// TIA Portal V15.1 export
// export: Created 2024-05-17T05:38:58.6337777Z, ExportSetting WithDefaults, DisplayName Totally Integrated Automation Portal, DisplayVersion V15.1 Update 5, DisplayName TIA Portal Openness, DisplayVersion V15.1 Update 5, DisplayName SINAMICS Startdrive Advanced, DisplayVersion V15.1, DisplayName G130, G150, S120, S150, SINAMICS MV, S210, DisplayVersion V15.1, DisplayName G110M, G120, G120C, G120D, G120P, DisplayVersion V15.1, DisplayName STEP 7 Professional, DisplayVersion V15.1 Update 5, DisplayName STEP 7 Safety, DisplayVersion V15.1, DisplayName WinCC Professional, DisplayVersion V15.1 Update 5, DisplayName SIMATIC Visualization Architect, DisplayVersion V15.1
FUNCTION "209230ZS01AEAK" : Void   // FC421, FBD
TITLE = 209230ZS01AEAK
{ S7_Optimized_Access := 'TRUE' }
AUTHOR : VCC
VERSION : 0.1
// stored: AutoNumber false, IsIECCheckEnabled false, SetENOAutomatically False, UDAEnableTagReadback false
   VAR_OUTPUT
      O_AlarmA : Bool;   // Alarm A
      O_AlarmB : Bool;   // Alarm B
      O_AlarmC : Bool;   // Alarm C
      O_AlarmD : Bool;   // Alarm D
      O_AlarmABCondition : Bool;   // Alarm AB condition
      H_IAnim : Word;   // For animation of icon
   END_VAR
BEGIN

REGION Network 1: **** --------------------- AE01 --------------------- ****
END_REGION

REGION Network 2: **** 2.2 Alarms - Alarm generation **** AE01E3FS13 // CH1 - 24VDC Fuse - ModeZone230 - Switch / Busnode 230AX01 & 230AS10
   // 24VDC Fuse - ModeZone230 - Switch / Busnode 230AX01 & 230AS10
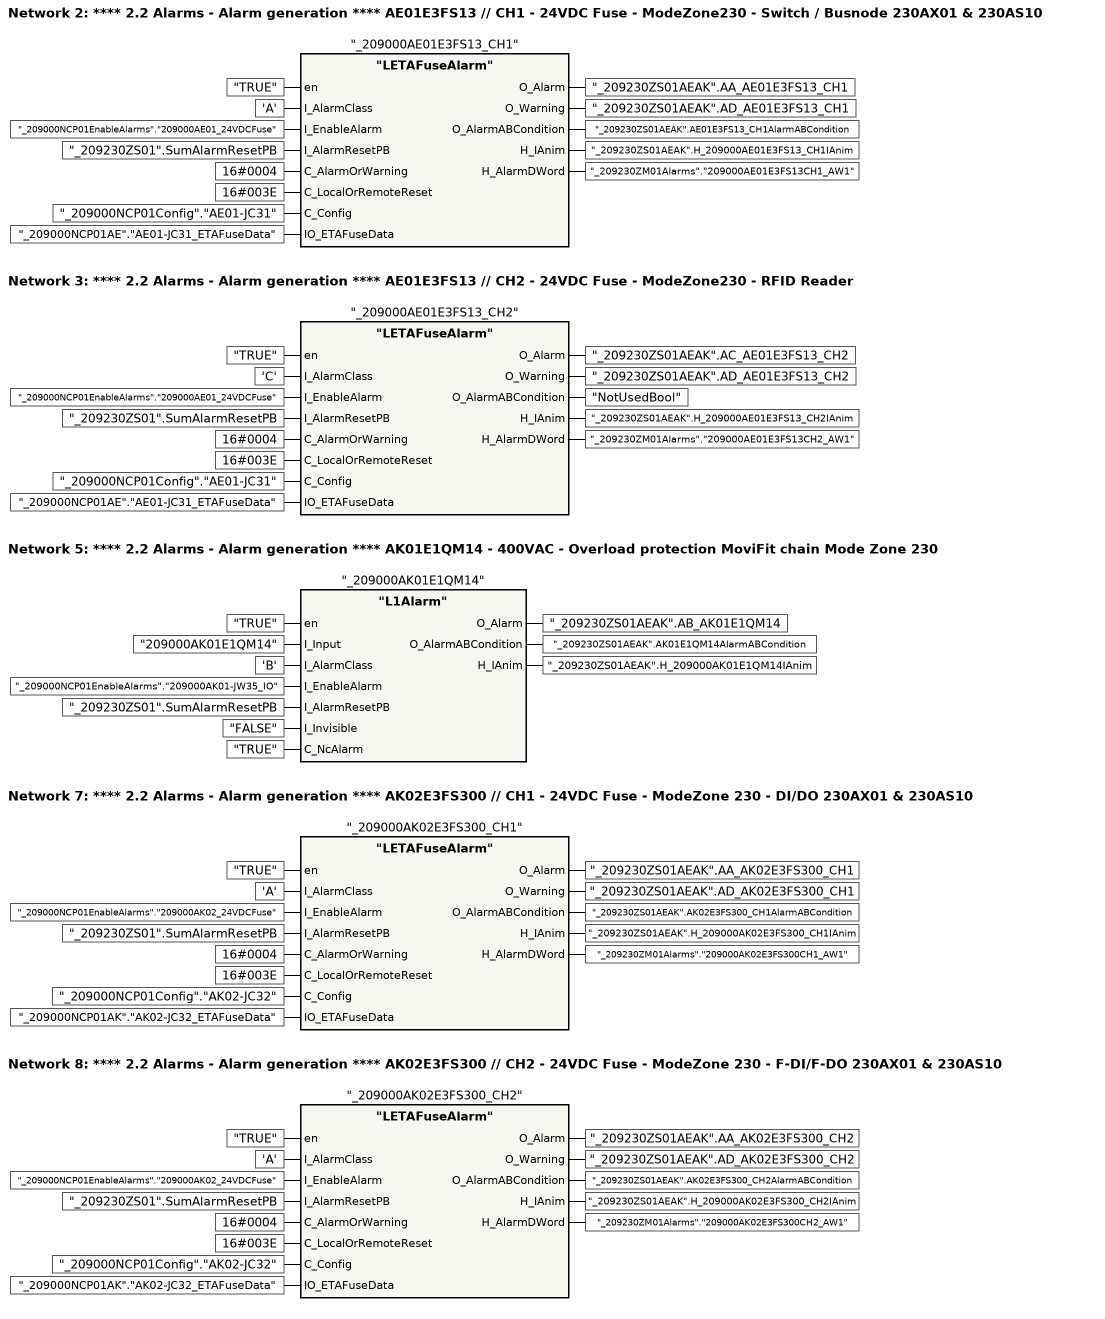
   IF "TRUE" THEN
       "_209000AE01E3FS13_CH1"(I_AlarmClass := 'A',   // "LETAFuseAlarm"
                               I_EnableAlarm := "_209000NCP01EnableAlarms"."209000AE01_24VDCFuse",
                               I_AlarmResetPB := "_209230ZS01".SumAlarmResetPB,
                               C_AlarmOrWarning := 16#0004,
                               C_LocalOrRemoteReset := 16#003E,
                               C_Config := "_209000NCP01Config"."AE01-JC31",
                               IO_ETAFuseData := "_209000NCP01AE"."AE01-JC31_ETAFuseData",
                               O_Alarm => "_209230ZS01AEAK".AA_AE01E3FS13_CH1,
                               O_Warning => "_209230ZS01AEAK".AD_AE01E3FS13_CH1,
                               O_AlarmABCondition => "_209230ZS01AEAK".AE01E3FS13_CH1AlarmABCondition,
                               H_IAnim => "_209230ZS01AEAK".H_209000AE01E3FS13_CH1IAnim,
                               H_AlarmDWord => "_209230ZM01Alarms"."209000AE01E3FS13CH1_AW1");
   END_IF;
END_REGION

REGION Network 3: **** 2.2 Alarms - Alarm generation **** AE01E3FS13 // CH2 - 24VDC Fuse - ModeZone230 - RFID Reader
   // 24VDC Fuse - ModeZone230 - RFID Reader
   IF "TRUE" THEN
       "_209000AE01E3FS13_CH2"(I_AlarmClass := 'C',   // "LETAFuseAlarm"
                               I_EnableAlarm := "_209000NCP01EnableAlarms"."209000AE01_24VDCFuse",
                               I_AlarmResetPB := "_209230ZS01".SumAlarmResetPB,
                               C_AlarmOrWarning := 16#0004,
                               C_LocalOrRemoteReset := 16#003E,
                               C_Config := "_209000NCP01Config"."AE01-JC31",
                               IO_ETAFuseData := "_209000NCP01AE"."AE01-JC31_ETAFuseData",
                               O_Alarm => "_209230ZS01AEAK".AC_AE01E3FS13_CH2,
                               O_Warning => "_209230ZS01AEAK".AD_AE01E3FS13_CH2,
                               O_AlarmABCondition => "NotUsedBool",
                               H_IAnim => "_209230ZS01AEAK".H_209000AE01E3FS13_CH2IAnim,
                               H_AlarmDWord => "_209230ZM01Alarms"."209000AE01E3FS13CH2_AW1");
   END_IF;
END_REGION

REGION Network 4: **** --------------------- AK01 --------------------- ****
END_REGION

REGION Network 5: **** 2.2 Alarms - Alarm generation **** AK01E1QM14 - 400VAC - Overload protection MoviFit chain Mode Zone 230
   // 400VAC - Overload protection MoviFit chain Mode Zone 230
   IF "TRUE" THEN
       "_209000AK01E1QM14"(I_Input := "209000AK01E1QM14",   // "L1Alarm"
                           I_AlarmClass := 'B',
                           I_EnableAlarm := "_209000NCP01EnableAlarms"."209000AK01-JW35_IO",
                           I_AlarmResetPB := "_209230ZS01".SumAlarmResetPB,
                           I_Invisible := "FALSE",
                           C_NcAlarm := "TRUE",
                           O_Alarm => "_209230ZS01AEAK".AB_AK01E1QM14,
                           O_AlarmABCondition => "_209230ZS01AEAK".AK01E1QM14AlarmABCondition,
                           H_IAnim => "_209230ZS01AEAK".H_209000AK01E1QM14IAnim);
   END_IF;
END_REGION

REGION Network 6: **** --------------------- AK02 --------------------- ****
END_REGION

REGION Network 7: **** 2.2 Alarms - Alarm generation **** AK02E3FS300 // CH1 - 24VDC Fuse - ModeZone 230 - DI/DO 230AX01 & 230AS10
   // 24VDC Fuse - ModeZone 230 - DI/DO 230AX01 & 230AS10
   IF "TRUE" THEN
       "_209000AK02E3FS300_CH1"(I_AlarmClass := 'A',   // "LETAFuseAlarm"
                               I_EnableAlarm := "_209000NCP01EnableAlarms"."209000AK02_24VDCFuse",
                               I_AlarmResetPB := "_209230ZS01".SumAlarmResetPB,
                               C_AlarmOrWarning := 16#0004,
                               C_LocalOrRemoteReset := 16#003E,
                               C_Config := "_209000NCP01Config"."AK02-JC32",
                               IO_ETAFuseData := "_209000NCP01AK"."AK02-JC32_ETAFuseData",
                               O_Alarm => "_209230ZS01AEAK".AA_AK02E3FS300_CH1,
                               O_Warning => "_209230ZS01AEAK".AD_AK02E3FS300_CH1,
                               O_AlarmABCondition => "_209230ZS01AEAK".AK02E3FS300_CH1AlarmABCondition,
                               H_IAnim => "_209230ZS01AEAK".H_209000AK02E3FS300_CH1IAnim,
                               H_AlarmDWord => "_209230ZM01Alarms"."209000AK02E3FS300CH1_AW1");
   END_IF;
END_REGION

REGION Network 8: **** 2.2 Alarms - Alarm generation **** AK02E3FS300 // CH2 - 24VDC Fuse - ModeZone 230 - F-DI/F-DO 230AX01 & 230AS10
   // 24VDC Fuse - ModeZone 230 - F-DI/F-DO 230AX01 & 230AS10
   IF "TRUE" THEN
       "_209000AK02E3FS300_CH2"(I_AlarmClass := 'A',   // "LETAFuseAlarm"
                               I_EnableAlarm := "_209000NCP01EnableAlarms"."209000AK02_24VDCFuse",
                               I_AlarmResetPB := "_209230ZS01".SumAlarmResetPB,
                               C_AlarmOrWarning := 16#0004,
                               C_LocalOrRemoteReset := 16#003E,
                               C_Config := "_209000NCP01Config"."AK02-JC32",
                               IO_ETAFuseData := "_209000NCP01AK"."AK02-JC32_ETAFuseData",
                               O_Alarm => "_209230ZS01AEAK".AA_AK02E3FS300_CH2,
                               O_Warning => "_209230ZS01AEAK".AD_AK02E3FS300_CH2,
                               O_AlarmABCondition => "_209230ZS01AEAK".AK02E3FS300_CH2AlarmABCondition,
                               H_IAnim => "_209230ZS01AEAK".H_209000AK02E3FS300_CH2IAnim,
                               H_AlarmDWord => "_209230ZM01Alarms"."209000AK02E3FS300CH2_AW1");
   END_IF;
END_REGION

REGION Network 9: **** 2.2 Alarms - Alarm generation **** AK02E3FS301 // CH1 - 24VDC Fuse - ModeZone 230 - Doorlock
   // 24VDC Fuse - ModeZone 230 - Doorlock
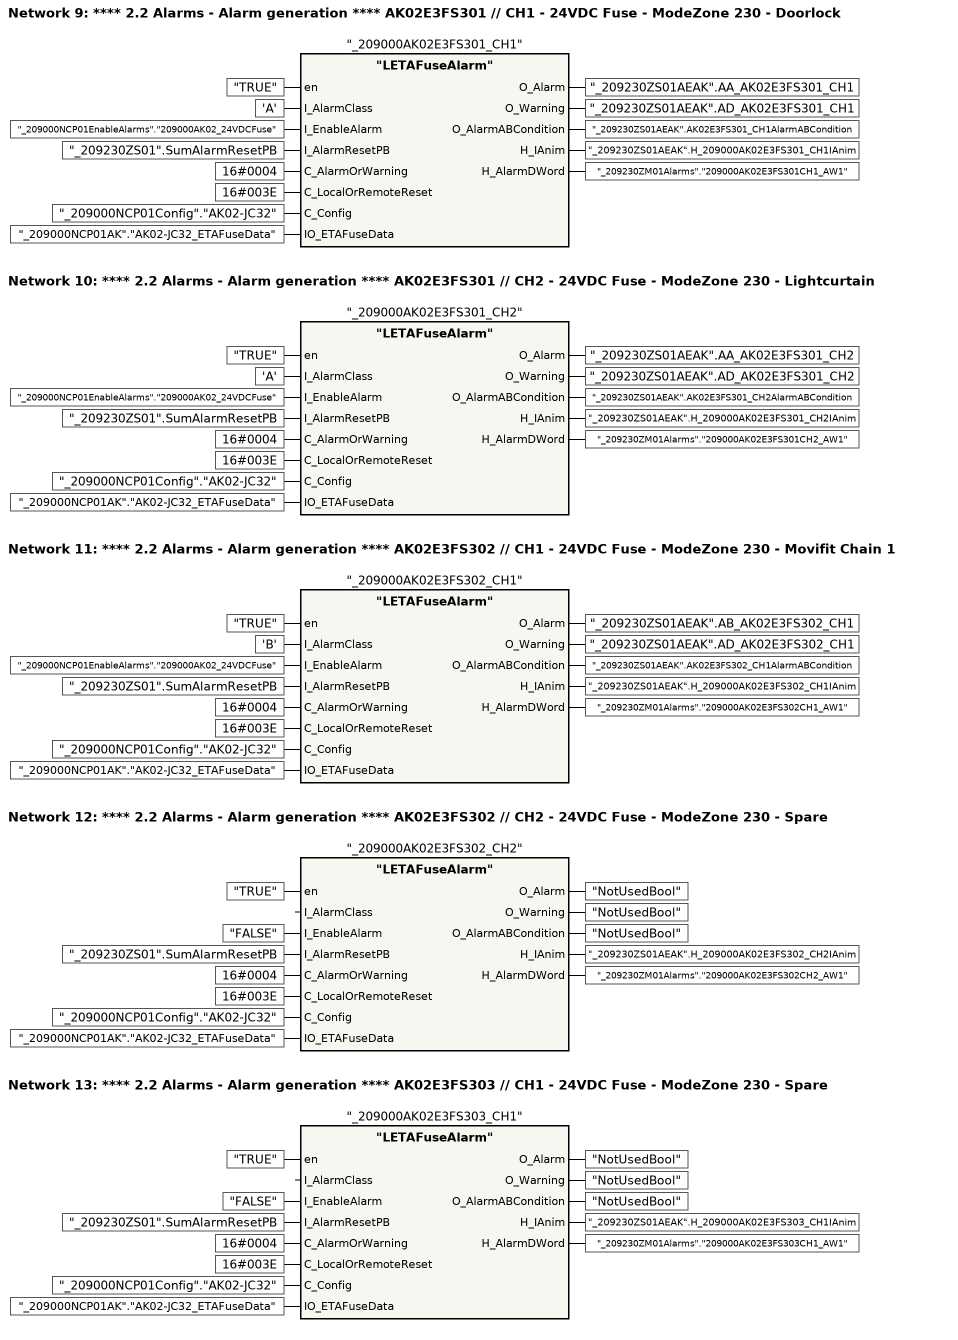
   IF "TRUE" THEN
       "_209000AK02E3FS301_CH1"(I_AlarmClass := 'A',   // "LETAFuseAlarm"
                               I_EnableAlarm := "_209000NCP01EnableAlarms"."209000AK02_24VDCFuse",
                               I_AlarmResetPB := "_209230ZS01".SumAlarmResetPB,
                               C_AlarmOrWarning := 16#0004,
                               C_LocalOrRemoteReset := 16#003E,
                               C_Config := "_209000NCP01Config"."AK02-JC32",
                               IO_ETAFuseData := "_209000NCP01AK"."AK02-JC32_ETAFuseData",
                               O_Alarm => "_209230ZS01AEAK".AA_AK02E3FS301_CH1,
                               O_Warning => "_209230ZS01AEAK".AD_AK02E3FS301_CH1,
                               O_AlarmABCondition => "_209230ZS01AEAK".AK02E3FS301_CH1AlarmABCondition,
                               H_IAnim => "_209230ZS01AEAK".H_209000AK02E3FS301_CH1IAnim,
                               H_AlarmDWord => "_209230ZM01Alarms"."209000AK02E3FS301CH1_AW1");
   END_IF;
END_REGION

REGION Network 10: **** 2.2 Alarms - Alarm generation **** AK02E3FS301 // CH2 - 24VDC Fuse - ModeZone 230 - Lightcurtain
   // 24VDC Fuse - ModeZone 230 - Lightcurtain
   IF "TRUE" THEN
       "_209000AK02E3FS301_CH2"(I_AlarmClass := 'A',   // "LETAFuseAlarm"
                               I_EnableAlarm := "_209000NCP01EnableAlarms"."209000AK02_24VDCFuse",
                               I_AlarmResetPB := "_209230ZS01".SumAlarmResetPB,
                               C_AlarmOrWarning := 16#0004,
                               C_LocalOrRemoteReset := 16#003E,
                               C_Config := "_209000NCP01Config"."AK02-JC32",
                               IO_ETAFuseData := "_209000NCP01AK"."AK02-JC32_ETAFuseData",
                               O_Alarm => "_209230ZS01AEAK".AA_AK02E3FS301_CH2,
                               O_Warning => "_209230ZS01AEAK".AD_AK02E3FS301_CH2,
                               O_AlarmABCondition => "_209230ZS01AEAK".AK02E3FS301_CH2AlarmABCondition,
                               H_IAnim => "_209230ZS01AEAK".H_209000AK02E3FS301_CH2IAnim,
                               H_AlarmDWord => "_209230ZM01Alarms"."209000AK02E3FS301CH2_AW1");
   END_IF;
END_REGION

REGION Network 11: **** 2.2 Alarms - Alarm generation **** AK02E3FS302 // CH1 - 24VDC Fuse - ModeZone 230 - Movifit Chain 1
   // 24VDC Fuse - ModeZone 230 - Movifit Chain 1
   IF "TRUE" THEN
       "_209000AK02E3FS302_CH1"(I_AlarmClass := 'B',   // "LETAFuseAlarm"
                               I_EnableAlarm := "_209000NCP01EnableAlarms"."209000AK02_24VDCFuse",
                               I_AlarmResetPB := "_209230ZS01".SumAlarmResetPB,
                               C_AlarmOrWarning := 16#0004,
                               C_LocalOrRemoteReset := 16#003E,
                               C_Config := "_209000NCP01Config"."AK02-JC32",
                               IO_ETAFuseData := "_209000NCP01AK"."AK02-JC32_ETAFuseData",
                               O_Alarm => "_209230ZS01AEAK".AB_AK02E3FS302_CH1,
                               O_Warning => "_209230ZS01AEAK".AD_AK02E3FS302_CH1,
                               O_AlarmABCondition => "_209230ZS01AEAK".AK02E3FS302_CH1AlarmABCondition,
                               H_IAnim => "_209230ZS01AEAK".H_209000AK02E3FS302_CH1IAnim,
                               H_AlarmDWord => "_209230ZM01Alarms"."209000AK02E3FS302CH1_AW1");
   END_IF;
END_REGION

REGION Network 12: **** 2.2 Alarms - Alarm generation **** AK02E3FS302 // CH2 - 24VDC Fuse - ModeZone 230 - Spare
   // 24VDC Fuse - ModeZone 230 - Spare
   IF "TRUE" THEN
       "_209000AK02E3FS302_CH2"(I_EnableAlarm := "FALSE",   // "LETAFuseAlarm"
                               I_AlarmResetPB := "_209230ZS01".SumAlarmResetPB,
                               C_AlarmOrWarning := 16#0004,
                               C_LocalOrRemoteReset := 16#003E,
                               C_Config := "_209000NCP01Config"."AK02-JC32",
                               IO_ETAFuseData := "_209000NCP01AK"."AK02-JC32_ETAFuseData",
                               O_Alarm => "NotUsedBool",
                               O_Warning => "NotUsedBool",
                               O_AlarmABCondition => "NotUsedBool",
                               H_IAnim => "_209230ZS01AEAK".H_209000AK02E3FS302_CH2IAnim,
                               H_AlarmDWord => "_209230ZM01Alarms"."209000AK02E3FS302CH2_AW1");
   END_IF;
END_REGION

REGION Network 13: **** 2.2 Alarms - Alarm generation **** AK02E3FS303 // CH1 - 24VDC Fuse - ModeZone 230 - Spare
   // 24VDC Fuse - ModeZone 230 - Spare
   IF "TRUE" THEN
       "_209000AK02E3FS303_CH1"(I_EnableAlarm := "FALSE",   // "LETAFuseAlarm"
                               I_AlarmResetPB := "_209230ZS01".SumAlarmResetPB,
                               C_AlarmOrWarning := 16#0004,
                               C_LocalOrRemoteReset := 16#003E,
                               C_Config := "_209000NCP01Config"."AK02-JC32",
                               IO_ETAFuseData := "_209000NCP01AK"."AK02-JC32_ETAFuseData",
                               O_Alarm => "NotUsedBool",
                               O_Warning => "NotUsedBool",
                               O_AlarmABCondition => "NotUsedBool",
                               H_IAnim => "_209230ZS01AEAK".H_209000AK02E3FS303_CH1IAnim,
                               H_AlarmDWord => "_209230ZM01Alarms"."209000AK02E3FS303CH1_AW1");
   END_IF;
END_REGION

REGION Network 14: **** 2.2 Alarms - Alarm generation **** AK02E3FS303 // CH2 - 24VDC Fuse - ModeZone 230 - Spare
   // 24VDC Fuse - ModeZone 230 - Spare
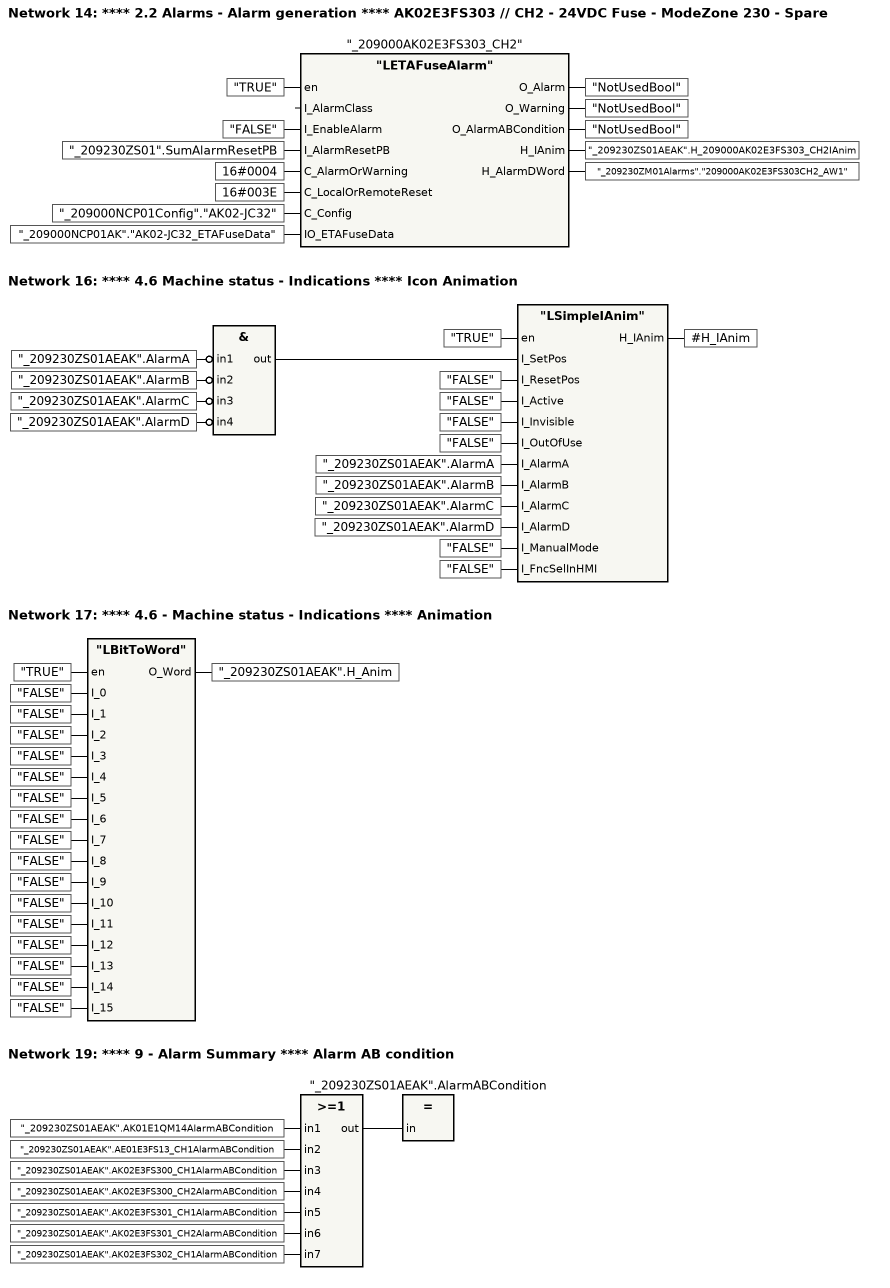
   IF "TRUE" THEN
       "_209000AK02E3FS303_CH2"(I_EnableAlarm := "FALSE",   // "LETAFuseAlarm"
                               I_AlarmResetPB := "_209230ZS01".SumAlarmResetPB,
                               C_AlarmOrWarning := 16#0004,
                               C_LocalOrRemoteReset := 16#003E,
                               C_Config := "_209000NCP01Config"."AK02-JC32",
                               IO_ETAFuseData := "_209000NCP01AK"."AK02-JC32_ETAFuseData",
                               O_Alarm => "NotUsedBool",
                               O_Warning => "NotUsedBool",
                               O_AlarmABCondition => "NotUsedBool",
                               H_IAnim => "_209230ZS01AEAK".H_209000AK02E3FS303_CH2IAnim,
                               H_AlarmDWord => "_209230ZM01Alarms"."209000AK02E3FS303CH2_AW1");
   END_IF;
END_REGION

REGION Network 15: **** -------------------------------------------------- ****
END_REGION

REGION Network 16: **** 4.6 Machine status - Indications **** Icon Animation
   // Animation for icon
   IF "TRUE" THEN
       "LSimpleIAnim"(I_SetPos := NOT "_209230ZS01AEAK".AlarmA AND NOT "_209230ZS01AEAK".AlarmB AND NOT "_209230ZS01AEAK".AlarmC AND NOT "_209230ZS01AEAK".AlarmD,
                      I_ResetPos := "FALSE",
                      I_Active := "FALSE",
                      I_Invisible := "FALSE",
                      I_OutOfUse := "FALSE",
                      I_AlarmA := "_209230ZS01AEAK".AlarmA,
                      I_AlarmB := "_209230ZS01AEAK".AlarmB,
                      I_AlarmC := "_209230ZS01AEAK".AlarmC,
                      I_AlarmD := "_209230ZS01AEAK".AlarmD,
                      I_ManualMode := "FALSE",
                      I_FncSelInHMI := "FALSE",
                      H_IAnim => #H_IAnim);
   END_IF;
END_REGION

REGION Network 17: **** 4.6 - Machine status - Indications **** Animation
   // Animation
   IF "TRUE" THEN
       "LBitToWord"(I_0 := "FALSE",
                    I_1 := "FALSE",
                    I_2 := "FALSE",
                    I_3 := "FALSE",
                    I_4 := "FALSE",
                    I_5 := "FALSE",
                    I_6 := "FALSE",
                    I_7 := "FALSE",
                    I_8 := "FALSE",
                    I_9 := "FALSE",
                    I_10 := "FALSE",
                    I_11 := "FALSE",
                    I_12 := "FALSE",
                    I_13 := "FALSE",
                    I_14 := "FALSE",
                    I_15 := "FALSE",
                    O_Word => "_209230ZS01AEAK".H_Anim);
   END_IF;
END_REGION

NETWORK
TITLE = **** 4.6 - Machine Status - Indications **** Animation DB number
// DB number
      OPN   "_209230ZS01AEAK";
      L     DBNO;
      T     "_209230ZS01AEAK".H_DBnr;

REGION Network 19: **** 9 - Alarm Summary **** Alarm AB condition
   // Alarm AB condition
   "_209230ZS01AEAK".AlarmABCondition := "_209230ZS01AEAK".AK01E1QM14AlarmABCondition OR "_209230ZS01AEAK".AE01E3FS13_CH1AlarmABCondition OR "_209230ZS01AEAK".AK02E3FS300_CH1AlarmABCondition OR "_209230ZS01AEAK".AK02E3FS300_CH2AlarmABCondition OR "_209230ZS01AEAK".AK02E3FS301_CH1AlarmABCondition OR "_209230ZS01AEAK".AK02E3FS301_CH2AlarmABCondition OR "_209230ZS01AEAK".AK02E3FS302_CH1AlarmABCondition;
END_REGION

REGION Network 20: **** 9 - Alarm Summary **** Alarm A
   // Summary of alarms A
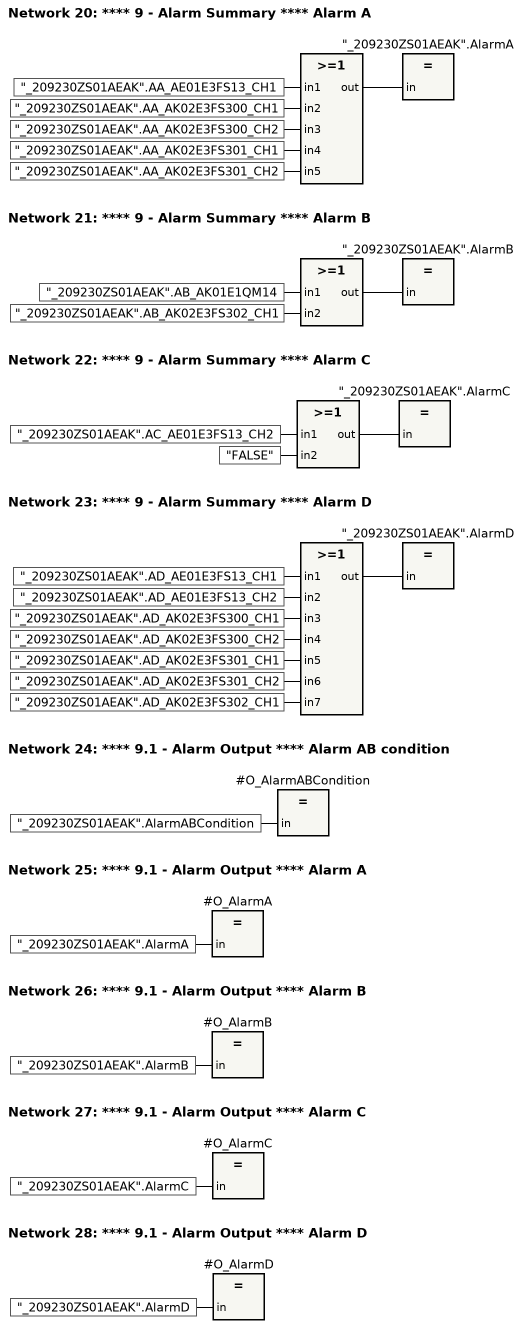
   "_209230ZS01AEAK".AlarmA := "_209230ZS01AEAK".AA_AE01E3FS13_CH1 OR "_209230ZS01AEAK".AA_AK02E3FS300_CH1 OR "_209230ZS01AEAK".AA_AK02E3FS300_CH2 OR "_209230ZS01AEAK".AA_AK02E3FS301_CH1 OR "_209230ZS01AEAK".AA_AK02E3FS301_CH2;
END_REGION

REGION Network 21: **** 9 - Alarm Summary **** Alarm B
   // Summary of alarms B
   "_209230ZS01AEAK".AlarmB := "_209230ZS01AEAK".AB_AK01E1QM14 OR "_209230ZS01AEAK".AB_AK02E3FS302_CH1;
END_REGION

REGION Network 22: **** 9 - Alarm Summary **** Alarm C
   // Summary of alarms C
   "_209230ZS01AEAK".AlarmC := "_209230ZS01AEAK".AC_AE01E3FS13_CH2 OR "FALSE";
END_REGION

REGION Network 23: **** 9 - Alarm Summary **** Alarm D
   // Summary of alarms D
   "_209230ZS01AEAK".AlarmD := "_209230ZS01AEAK".AD_AE01E3FS13_CH1 OR "_209230ZS01AEAK".AD_AE01E3FS13_CH2 OR "_209230ZS01AEAK".AD_AK02E3FS300_CH1 OR "_209230ZS01AEAK".AD_AK02E3FS300_CH2 OR "_209230ZS01AEAK".AD_AK02E3FS301_CH1 OR "_209230ZS01AEAK".AD_AK02E3FS301_CH2 OR "_209230ZS01AEAK".AD_AK02E3FS302_CH1;
END_REGION

REGION Network 24: **** 9.1 - Alarm Output **** Alarm AB condition
   // Alarm AB condition
   #O_AlarmABCondition := "_209230ZS01AEAK".AlarmABCondition;
END_REGION

REGION Network 25: **** 9.1 - Alarm Output **** Alarm A
   // Summary of alarms A
   #O_AlarmA := "_209230ZS01AEAK".AlarmA;
END_REGION

REGION Network 26: **** 9.1 - Alarm Output **** Alarm B
   // Summary of alarms B
   #O_AlarmB := "_209230ZS01AEAK".AlarmB;
END_REGION

REGION Network 27: **** 9.1 - Alarm Output **** Alarm C
   // Summary of alarms C
   #O_AlarmC := "_209230ZS01AEAK".AlarmC;
END_REGION

REGION Network 28: **** 9.1 - Alarm Output **** Alarm D
   // Summary of alarms D
   #O_AlarmD := "_209230ZS01AEAK".AlarmD;
END_REGION

REGION Network 29: **** 9.2 - Alarm DWord**** Alarm To DWord
   // Alarm Word
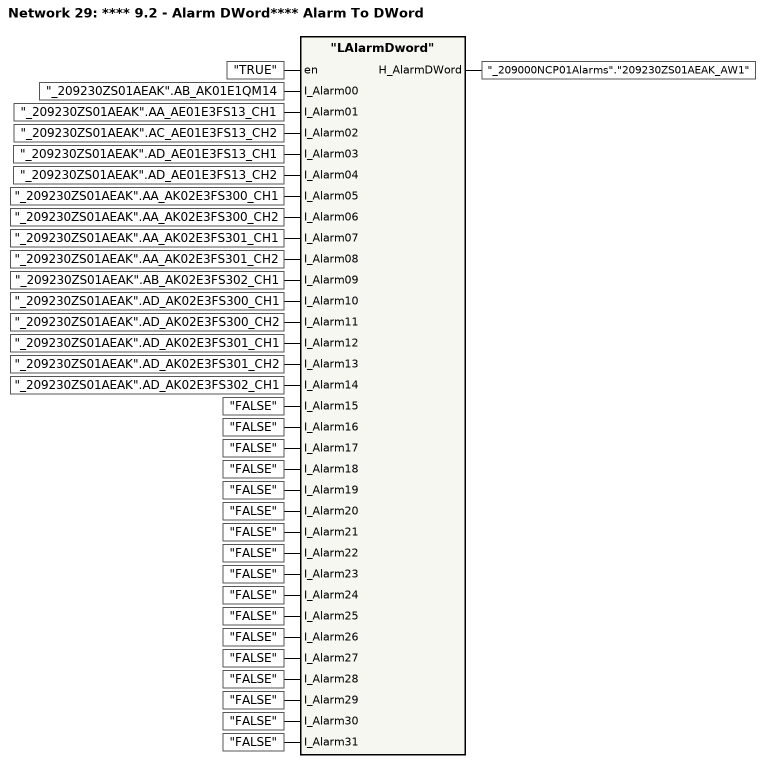
   IF "TRUE" THEN
       "LAlarmDword"(I_Alarm00 := "_209230ZS01AEAK".AB_AK01E1QM14,
                     I_Alarm01 := "_209230ZS01AEAK".AA_AE01E3FS13_CH1,
                     I_Alarm02 := "_209230ZS01AEAK".AC_AE01E3FS13_CH2,
                     I_Alarm03 := "_209230ZS01AEAK".AD_AE01E3FS13_CH1,
                     I_Alarm04 := "_209230ZS01AEAK".AD_AE01E3FS13_CH2,
                     I_Alarm05 := "_209230ZS01AEAK".AA_AK02E3FS300_CH1,
                     I_Alarm06 := "_209230ZS01AEAK".AA_AK02E3FS300_CH2,
                     I_Alarm07 := "_209230ZS01AEAK".AA_AK02E3FS301_CH1,
                     I_Alarm08 := "_209230ZS01AEAK".AA_AK02E3FS301_CH2,
                     I_Alarm09 := "_209230ZS01AEAK".AB_AK02E3FS302_CH1,
                     I_Alarm10 := "_209230ZS01AEAK".AD_AK02E3FS300_CH1,
                     I_Alarm11 := "_209230ZS01AEAK".AD_AK02E3FS300_CH2,
                     I_Alarm12 := "_209230ZS01AEAK".AD_AK02E3FS301_CH1,
                     I_Alarm13 := "_209230ZS01AEAK".AD_AK02E3FS301_CH2,
                     I_Alarm14 := "_209230ZS01AEAK".AD_AK02E3FS302_CH1,
                     I_Alarm15 := "FALSE",
                     I_Alarm16 := "FALSE",
                     I_Alarm17 := "FALSE",
                     I_Alarm18 := "FALSE",
                     I_Alarm19 := "FALSE",
                     I_Alarm20 := "FALSE",
                     I_Alarm21 := "FALSE",
                     I_Alarm22 := "FALSE",
                     I_Alarm23 := "FALSE",
                     I_Alarm24 := "FALSE",
                     I_Alarm25 := "FALSE",
                     I_Alarm26 := "FALSE",
                     I_Alarm27 := "FALSE",
                     I_Alarm28 := "FALSE",
                     I_Alarm29 := "FALSE",
                     I_Alarm30 := "FALSE",
                     I_Alarm31 := "FALSE",
                     H_AlarmDWord => "_209000NCP01Alarms"."209230ZS01AEAK_AW1");
   END_IF;
END_REGION
END_FUNCTION
